// TwinCAT 3 PLC project plc_tmo_hutch_vac_fs
// ProgramVersion: 3.1.4023.0
// libraries:
//   LCLS General, * (SLAC)
//   LCLS Vacuum, * (SLAC - LCLS)
//   PMPS, * (SLAC - LCLS)
//   Tc2_Standard, * (Beckhoff Automation GmbH)
//   Tc2_System, * (Beckhoff Automation GmbH)
//   Tc3_Module, * (Beckhoff Automation GmbH)
// project tree:
//   GVLs/ GVL_FSV_PMPS.TcGVL, GVL_FS_Devices.TcGVL
//   / PlcTask.TcTTO
//   POUs/ MAIN.TcPOU
// (motion and I/O tree: see PLC project plc_tmo_hutch_vac)
// real-time tasks:
//   TASK PlcTask: cycle T#10ms, priority 20, ADS port 350
//   TASK ComTask: cycle T#3ms, priority 21, ADS port 351
//   TASK FSVTask: cycle T#1ms, priority 1, ADS port 352
// variable links:
//   plc_tmo_hutch_vac_fs/plc_tmo_hutch_vac_fs Instance <-> Device 1 (EtherCAT)/TMO_K4S2_DRL_01 (EK1100)/K4S2_01_E1_VFS (EL1004)
//     PlcTask Inputs/GVL_FS_Devices.MR3K4_KBO_VFS_1.i_xClsLS <-> Channel 1/Input
//     PlcTask Inputs/GVL_FS_Devices.MR3K4_KBO_VFS_1.i_xOpnLS <-> Channel 2/Input
//   plc_tmo_hutch_vac_fs/plc_tmo_hutch_vac_fs Instance <-> Device 1 (EtherCAT)/TMO_K4S2_DRL_01 (EK1100)/K4S2_01_E3_VFS (EL2202)
//     PlcTask Outputs/GVL_FS_Devices.MR3K4_KBO_VFS_1.q_xClose_A <-> Channel 1/Output
//     PlcTask Outputs/GVL_FS_Devices.MR3K4_KBO_VFS_1.q_xClose_B <-> Channel 2/Output
//   plc_tmo_hutch_vac_fs/plc_tmo_hutch_vac_fs Instance <-> Device 1 (EtherCAT)/TMO_K4S2_DRL_01 (EK1100)/K4S2_01_E4_VFS (EL2202)
//     PlcTask Outputs/GVL_FS_Devices.MR3K4_KBO_VFS_1.q_xClose_C <-> Channel 1/Output
//     PlcTask Outputs/GVL_FS_Devices.MR3K4_KBO_VFS_1.q_xOPN_DO <-> Channel 2/Output
//   plc_tmo_hutch_vac_fs/plc_tmo_hutch_vac_fs Instance <-> Device 1 (EtherCAT)/TMO_K4S8_DRL_01 (EK1100)/K4S8_01_E1 (EL1004)
//     PlcTask Inputs/GVL_FS_Devices.MR4K4_KBO_VFS_1.i_xClsLS <-> Channel 1/Input
//     PlcTask Inputs/GVL_FS_Devices.MR4K4_KBO_VFS_1.i_xOpnLS <-> Channel 2/Input
//   plc_tmo_hutch_vac_fs/plc_tmo_hutch_vac_fs Instance <-> Device 1 (EtherCAT)/TMO_K4S8_DRL_01 (EK1100)/K4S8_01_E3 (EL2202)
//     PlcTask Outputs/GVL_FS_Devices.MR4K4_KBO_VFS_1.q_xClose_A <-> Channel 1/Output
//     PlcTask Outputs/GVL_FS_Devices.MR4K4_KBO_VFS_1.q_xClose_B <-> Channel 2/Output
//   plc_tmo_hutch_vac_fs/plc_tmo_hutch_vac_fs Instance <-> Device 1 (EtherCAT)/TMO_K4S8_DRL_01 (EK1100)/K4S8_01_E4 (EL2202)
//     PlcTask Outputs/GVL_FS_Devices.MR4K4_KBO_VFS_1.q_xClose_C <-> Channel 1/Output
//     PlcTask Outputs/GVL_FS_Devices.MR4K4_KBO_VFS_1.q_xOPN_DO <-> Channel 2/Output

CONFIGURATION plc_tmo_hutch_vac_fs
    RESOURCE PLC ON TwinCAT3
        TASK PlcTask(INTERVAL := T#12ms, PRIORITY := 21);
        PROGRAM MAIN WITH PlcTask : MAIN;
    END_RESOURCE
END_CONFIGURATION

// ---- GVLs/GVL_FSV_PMPS.TcGVL
VAR_GLOBAL

	
	{'attribute 'pytmc' := 'pv: TMO:VAC:FFO:03  '}
    //{attribute 'TcLinkTo' := '.q_xFastFaultOut:=TIIB[CX0_E1 (EL2202)]^Channel 2^Output'}
    g_FastFaultOutput3  :   FB_HardwareFFOutput;	//FFO for TV1K4-VFS-1
	
	
END_VAR

// ---- GVLs/GVL_FS_Devices.TcGVL
VAR_GLOBAL
    {attribute 'pytmc' := '
		pv: MR3K4:KBO:VFS_1
	'}
	{attribute 'TcLinkTo' := 	'
		.q_xClose_A	:=	TIIB[K4S2_01_E3_VFS (EL2202)]^Channel 1^Output;
		.q_xClose_B	:=	TIIB[K4S2_01_E3_VFS (EL2202)]^Channel 2^Output;
		.q_xClose_C	:=	TIIB[K4S2_01_E4_VFS (EL2202)]^Channel 1^Output;
		.q_xOPN_DO	:=	TIIB[K4S2_01_E4_VFS (EL2202)]^Channel 2^Output;
		.i_xClsLS	:=	TIIB[K4S2_01_E1_VFS (EL1004)]^Channel 1^Input;
		.i_xOpnLS	:=	TIIB[K4S2_01_E1_VFS (EL1004)]^Channel 2^Input;
		.i_xTrigger := 	'}
	MR3K4_KBO_VFS_1 : FB_VFS;
	
	{attribute 'pytmc' := '
		pv: MR3K4:KBO:VFS_1
	'}
	{attribute 'TcLinkTo' := 	'
		.q_xClose_A	:=	TIIB[K4S8_01_E3 (EL2202)]^Channel 1^Output;
		.q_xClose_B	:=	TIIB[K4S8_01_E3 (EL2202)]^Channel 2^Output;
		.q_xClose_C	:=	TIIB[K4S8_01_E4 (EL2202)]^Channel 1^Output;
		.q_xOPN_DO	:=	TIIB[K4S8_01_E4 (EL2202)]^Channel 2^Output;
		.i_xClsLS	:=	TIIB[K4S8_01_E1 (EL1004)]^Channel 1^Input;
		.i_xOpnLS	:=	TIIB[K4S8_01_E1 (EL1004)]^Channel 2^Input;
		.i_xTrigger := 	'}
	MR4K4_KBO_VFS_1 : FB_VFS;
END_VAR

// ---- POUs/MAIN.TcPOU
PROGRAM MAIN
VAR
END_VAR

MR3K4_KBO_VFS_1(
	i_xPMPS_OK:= TRUE, 
	i_xExt_OK:= TRUE, 
	i_sDevName:= 'MR3K4:KBO:VFS:1',
	io_fbFFHWO:= g_FastFaultOutput3
);

MR4K4_KBO_VFS_1(
	i_xPMPS_OK:= TRUE, 
	i_xExt_OK:= TRUE, 
	i_sDevName:= 'MR4K4:KBO:VFS:1',
	io_fbFFHWO:= g_FastFaultOutput3
);
(*FastFaultOuput*)	
g_FastFaultOutput3.Execute(bAutoReset:= TRUE);

END_PROGRAM
